ABB RobotStudio station: IndustrialFinal_1.rspag

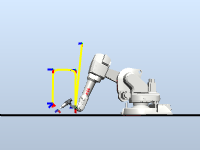
--- station ---
Station IndustrialFinal_1 (saved by RobotStudio 6.6.7624.115)
Controller IRB_1600_8kg_1.2m
  mechanical unit ROB_1: IRB1600_8_120__02, 6 joints, base frame (0, 0, 0) mm
Layout (positions relative to the parent item):
  - IRB1600_8_120__02 [mechanism, from Robots\IRB1600_8_120_G_02.rslib] at (0, 0, 0) mm; joint values [-0.0084, 1.2169, -0.0527, -0.0091, -1.1643, 0.0036] (rad or m)
  - MyTool [mechanism, from Training Objects\myTool.rslib] at (897.81, -6.97, 100) mm, rotated rx -170.3 ry 90 rz -170.3 deg
Attachment: MyTool is attached to IRB1600_8_120__02 / Link6
Targets, tools, work objects and paths stored in the station and not in the controller backup, written as RAPID:
! task T_ROB1
MODULE Module1
  CONST jointtarget Home_Pos:=[[0,0,0,0,0,0],[9E+09,9E+09,9E+09,9E+09,9E+09,9E+09]];
  CONST robtarget Coffee_Grab:=[[897.808,-6.966,100],[0.707106781,0,0.707106781,0],[-1,-1,0,1],[9E+09,9E+09,9E+09,9E+09,9E+09,9E+09]];
  CONST robtarget Coffee_Up:=[[897.808,-6.966,600],[0.707106781,0,0.707106781,0],[-1,-1,0,1],[9E+09,9E+09,9E+09,9E+09,9E+09,9E+09]];
  CONST robtarget Over_Cup:=[[1197.808,-6.966,600],[0.707106781,0,0.707106781,0],[-1,-1,0,1],[9E+09,9E+09,9E+09,9E+09,9E+09,9E+09]];
  CONST robtarget Ready_Pour:=[[1197.808,-6.966,150],[0.707106781,0,0.707106781,0],[-1,-1,0,1],[9E+09,9E+09,9E+09,9E+09,9E+09,9E+09]];
  CONST robtarget Pour:=[[1197.808,-6.966,150],[0.382683431,0,0.923879533,0],[-1,0,-1,0],[9E+09,9E+09,9E+09,9E+09,9E+09,9E+09]];
  PROC Path_20()
    MoveAbsJ Home_Pos,v1000,z100,tool0\WObj:=wobj0;
    MoveL Coffee_Grab,v1000,z100,tool0\WObj:=wobj0;
    MoveL Coffee_Up,v1000,z100,tool0\WObj:=wobj0;
    MoveL Over_Cup,v1000,z100,tool0\WObj:=wobj0;
    MoveL Ready_Pour,v1000,z100,tool0\WObj:=wobj0;
    MoveL Pour,v1000,z100,tool0\WObj:=wobj0;
    MoveL Ready_Pour,v1000,z100,tool0\WObj:=wobj0;
    MoveL Over_Cup,v1000,z100,tool0\WObj:=wobj0;
    MoveL Coffee_Up,v1000,z100,tool0\WObj:=wobj0;
    MoveL Coffee_Grab,v1000,z100,tool0\WObj:=wobj0;
  ENDPROC
ENDMODULE


--- Backups/IRB_1600_8kg_1.2m/RAPID/TASK1/PROGMOD/Module1.mod ---
MODULE Module1
    !***********************************************************
    !
    ! Module:  Module1
    !
    ! Description:
    !   <Insert description here>
    !
    ! Author: lgstuehrmann
    !
    ! Version: 1.0
    !
    !***********************************************************


    !***********************************************************
    !
    ! Procedure main
    !
    !   This is the entry point of your program
    !
    !***********************************************************
    PROC main()
        !Add your code here
    ENDPROC
ENDMODULE

--- Backups/IRB_1600_8kg_1.2m/RAPID/TASK1/SYSMOD/LINKEDM.sys ---
%%%
  VERSION:1
  LANGUAGE:ENGLISH
%%%

MODULE LINKEDM (SYSMODULE)

! FOLLOWER
!     Name of electronically linked follower axis used by operator at teach pendent.
      PERS string l_f_axis_name{5}       :=  ["",  "", "", "", ""];

!     Name of the mechanical unit for follower axis.
      PERS string l_f_mecunt_n{5}  :=  ["", "", "", "", ""];

!     Linked follower axis number in the mechanical unit (first axis in mech. unit is number 1).
      PERS num l_f_axis_no{5}      :=  [0,          0,   0,  0,  0];

! MASTER
!     Name of the mechanical unit for linked master axis.
      PERS string l_m_mecunt_n{5} :=  ["", "", "", "", ""];

!     Linked master axis number in the mechanical unit (first axis in mech. unit is number 1).
!     See axis number table in documentation for different master mechanical units.
      PERS num l_m_axis_no{5}     :=  [0,  0,  0,  0,  0];

! POSITION OFFSET
!     The increase of the allowed offset position between the master and follower
!     positions, used when starting AUTO mode. As soon as the offset is decreased
!     the old configurated parameter is used.
!     Example: 3 => the configurated value of allowed offset is increased 3 times.
      PERS num offset_ratio{5}       :=  [10,  10,   10,  10,  10];

! SPEED RATIO
!     Speed_ratio used in AUTO and JOG modes [ very_slow   slow    normal    fast]
!     Value 1 = max allowed manual speed.
      CONST num speed_ratio {20}      := [0.01, 0.01, 0.01, 0.01, 0.01,
                                          0.05, 0.05, 0.05, 0.05, 0.05,
                                          0.20, 0.20, 0.20, 0.20, 0.20,
                                          1.00, 1.00, 1.00, 1.00, 1.00];

! STEP SIZE
!     Displacement position used in JOG mode for each activation of positive or
!     negative movement.                  [very_short    short   normal   long]
!     Unit degees or meter.
      CONST num displacement {20}     := [0.001, 0.001, 0.001, 0.001, 0.001,
                                          0.005, 0.005, 0.005, 0.005, 0.005,
                                          0.020, 0.020, 0.020, 0.020, 0.020,
                                          0.100, 0.100, 0.100, 0.100, 0.100];


!-------------------------------------------------------------
 PROC Linked_m ()
      Linked_m_exe ;
 ENDPROC
ENDMODULE
